TYPE ST_Chamber1_ServiceCtrl :
STRUCT
	SpinAxisJogCW : ST_ServiceCtrl;
	SpinAxisMoveAbs : ST_ServiceCtrl;
	SpinAxisMoveVelCW	: ST_ServiceCtrl;
	LiftPinAxisMoveVelCW : ST_ServiceCtrl;
	LiftPinAxisMoveVelCCW : ST_ServiceCtrl;
	LiftPinAxisMoveAbs : ST_ServiceCtrl;
	
	DoorClose : ST_ServiceCtrl;
	DoorOpen : ST_ServiceCtrl;
	VacuumOn : ST_ServiceCtrl;
	VacuumOff : ST_ServiceCtrl;
	PreparePosition : ST_ServiceCtrl;
	Endpoint1PrepareSendWafer : ST_ServiceCtrl;
	SetMaterial : ST_ServiceCtrl;
END_STRUCT
END_TYPE

(* stored: Version 1.1.0.1, ProductVersion 3.1.4026.18
   DUT ST_Chamber1_ServiceCtrl: Id {ffd8beff-04a4-4f84-92ab-5776cc33b725} *)
